# EPICS StreamDevice protocol: LVREMOTE/LVREMOTE-IOC-01App/protocol/lvremote_string.proto
Terminator = CR LF;
path="%#/\//\\/";

getString {
    out "LVGET \${1}" ${path} ",\$2";
    in "%#s";
}
sendString {
    out "LVPUT \$1" ${path} ",\$2,%s";
    @init { getString; }
}
